INTERFACE iBase EXTENDS __SYSTEM.IQueryInterface

END_INTERFACE

(* stored: Version 1.1.0.1, ProductVersion 3.1.4026.18
   Itf iBase: Id {b10eef02-8809-0e7e-13cf-6334935f2a70} *)
